(* CODESYS project PFC_can_J1939_localport_v0.0.1.ecp

Project tree, tasks and I/O mapping:
  Controller_1 : 750-8203 PFC200 2ETH CAN, WAGO, order no. 0750-8203, version 5.11.1.16
    application Application
      libraries: ; WagoAppCanLayer2, * (WAGO); WagoSysErrorBase, * (WAGO); WagoSysFieldbus_75x_658, 1.6.0.4 (WAGO)
      task PLC_Task (cyclic, interval t#50ms, priority 15) calls PLC_PRG
      global variables GVL
      program PLC_PRG [ST]
    DeviceAdapter
    Kbus : Kbus, WAGO, version 1.4.0.2
        unmapped channels: K-BUS diagnostics
      _8DIO_24_VDC_0_5A : 0750-1506, WAGO, order no. 0750-1506, version 0.0.0.11
          unmapped channels: _IN, _OUT
        DeviceAdapter
    MODBUS
      MODBUS : MODBUS, WAGO, order no. n/a, version 1.1.1.15
    CANbus
      WAGO_CAN_LAYER2_DEVICE : WAGO CAN Layer2 Device, WAGO, version 3.5.4.9
  libraries: VisuSymbols, 3.5.10.0 (System); WagoVisuIcons, 1.0.0.8 (WAGO)
  data type CAN_Data
  text list GlobalTextList
*)

// CAN_Data
TYPE CAN_Data :
STRUCT
	ID		: DWORD;
	Data	: ARRAY[0..7]OF BYTE;
END_STRUCT
END_TYPE

// Controller_1/Application/GVL
{attribute 'qualified_only'}
VAR_GLOBAL
	xFirstScan		: BOOL := TRUE;
	wCanRx29BitAllMsgCounter : WORD;
	myTIme: INT;
END_VAR

// Controller_1/Application/PLC_PRG
PROGRAM PLC_PRG
VAR
	(* LOCAL CAN PORT reading J1939
	written by: Jesse Cox WAGO USA jesse.cox@wago.com *)
	
	// functional vars
	rtClosePortTrig		: R_TRIG;
	
	// CAN data vars
	BufferIndex			: INT := 0;
	i					: INT;
	myCanData			: ARRAY[0..iMaxCanBuffer] OF CAN_Data;
	myCanMsgCount		: WORD;
	rtReadIntoBuffer	: R_TRIG;
	
	// open block vars
	fbCanOpenPort		: FbCanL2Open;
	xCanPortEnable		: BOOL;
	udiCanPortBaud		: UDINT := 500000;
	dwCanPortFlags		: DWORD := 15;
	xCanPortOpenIsValid	: BOOL;
	xCanPortOpenIsBusy	: BOOL;
	xCanPortOpenError	: BOOL;
	oCanPortOpenStatus	: WagoSysErrorBase.FbResult;
	
	//  close block vars
	fbCanPortClose		: FbCanL2Close;
	xCanPortCloseEnable	: BOOL;
	xCanPortCloseDone	: BOOL;
	xCanPortCloseError	: BOOL;
	xCanPortCloseBusy	: BOOL;
	oCanPortCloseStatus	: WagoSysErrorBase.FbResult;
	
	// Rx vars header
	fbCanRx29Bit		: FbCanRx29BitFrame;
	xCanRx29BitEnable	: BOOL;
	xCanRx29BitBufferEnable: BOOL;
	dwCanRx29BitID		: DWORD := 16#1CFF0080;
	xCanRx29BitTrigger	: BOOL;
	xCanRx29BitIsValid	: BOOL;
	xCanRx29BitError	: BOOL;
	xCanRx29BitBusy		: BOOL;
	oCanRx29BitStatus	: WagoSysErrorBase.FbResult;
	wCanRx29BitMsgCounter: WORD;
	wCanRx29BitFrames	: WORD;
	xCanRx29BitRTR		: BOOL;
	bCanRx29BitBytes	: BYTE;
	aCanRx29BitInBuffer	: ARRAY [1..8] OF BYTE;
	
	// Rx All vars
	fbCanRx29BitAll		: FbCanRx29BitFrameAll;
	
	xCanRx29BitAllEnable: BOOL;
	xCanRx29BitAllBufferEnable: BOOL := TRUE;;
	xCanRx29BitAllTrigger: BOOL;
	xCanRx29BitAllIsValid: BOOL;
	xCanRx29BitAllError: BOOL;
	xCanRx29BitAllBusy: BOOL;
	oCanRx29BitAllStatus: WagoSysErrorBase.FbResult;
	wCanRx29BitAllFrames: WORD;
	xCanRx29BitAllRTR: BOOL;
	bCanRx29BitAllBytes: BYTE;
	aCanRx29BitAllInBuffer: ARRAY [1..8] OF BYTE;
	dwCanRx29BitAllInDataID: DWORD;
	
	// count valid flags
	rtValid					: R_TRIG;
	wValidJunk				: WORD;
	
	wJunk: INT;
	xCountUp: BOOL;
END_VAR

VAR CONSTANT
	iMaxCanBuffer	: INT := 500;
END_VAR


xCanPortEnable := TRUE;

// open the CAN port on the CAN Gateway module
fbCanOpenPort(
	xEnable:= xCanPortEnable, 
	I_Port:= IoConfig_Globals.WAGO_CAN_LAYER2_DEVICE, 
	udiBaudrate:= udiCanPortBaud, 
	dwFlags:= dwCanPortFlags, 
	dwPara:= , 
	xValid=> xCanPortOpenIsValid, 
	xBusy=> xCanPortOpenIsBusy, 
	xError=> xCanPortOpenError, 
	oStatus=> oCanPortOpenStatus);
	
// enable the read fb when the CAN port is open
xCanRx29BitAllEnable := xCanPortOpenIsValid;
	
// close the CAN port
fbCanPortClose(
	xExecute:= xCanPortCloseEnable, 
	I_Port:= IoConfig_Globals.WAGO_CAN_LAYER2_DEVICE, 
	xDone=> xCanPortCloseDone, 
	xError=> xCanPortCloseError, 
	xBusy=> xCanPortCloseBusy, 
	oStatus=> oCanPortCloseStatus);	
	
// read the Rx regs
fbCanRx29Bit(
	xEnable:= xCanRx29BitEnable, 
	I_Port:= IoConfig_Globals.WAGO_CAN_LAYER2_DEVICE, 
	xBufferMode:= xCanRx29BitBufferEnable, 
	dwCanId:= dwCanRx29BitID, 
	xRxTrigger:= xCanRx29BitTrigger, 
	xValid=> xCanRx29BitIsValid, 
	xError=> xCanRx29BitError, 
	xBusy=> xCanRx29BitBusy, 
	oStatus=> oCanRx29BitStatus, 
	wCounter=> wCanRx29BitMsgCounter, 
	wFrames=> wCanRx29BitFrames, 
	xRtrFrame=> xCanRx29BitRTR, 
	bRxNBytes=> bCanRx29BitBytes, 
	aRxBuffer=> aCanRx29BitInBuffer);
	
	rtValid(CLK := NOT xCanRx29BitAllIsValid);
	IF rtValid.Q THEN
		wValidJunk := wValidJunk + 1;
	END_IF
	
fbCanRx29BitAll(
	xEnable:= xCanRx29BitAllEnable, 
	I_Port:= IoConfig_Globals.WAGO_CAN_LAYER2_DEVICE, 
	xBufferMode:= xCanRx29BitAllBufferEnable, 
	xRxTrigger:= xCanRx29BitAllTrigger, 
	xValid=> xCanRx29BitAllIsValid, 
	xError=> xCanRx29BitAllError, 
	xBusy=> xCanRx29BitAllBusy, 
	oStatus=> oCanRx29BitAllStatus, 
	wCounter=> GVL.wCanRx29BitAllMsgCounter, 
	wFrames=> wCanRx29BitAllFrames, 
	xRtrFrame=> xCanRx29BitAllRTR, 
	bRxNBytes=> bCanRx29BitAllBytes, 
	aRxBuffer=> aCanRx29BitAllInBuffer, 
	dwRxId=> dwCanRx29BitAllInDataID);
	
	//process the incoming CAN data
IF xCanRx29BitAllEnable AND ((GVL.wCanRx29BitAllMsgCounter <> myCanMsgCount) OR (wCanRx29BitAllFrames > 0)) THEN
	xCanRx29BitAllTrigger := TRUE;
	myCanMsgCount := GVL.wCanRx29BitAllMsgCounter;
END_IF
rtReadIntoBuffer(CLK:= NOT xCanRx29BitAllTrigger);
IF rtReadIntoBuffer.Q THEN
		myCanData[GVL.wCanRx29BitAllMsgCounter].ID := dwCanRx29BitAllInDataID;
		myCanData[GVL.wCanRx29BitAllMsgCounter].Data := aCanRx29BitAllInBuffer;
END_IF

END_PROGRAM
